# EPICS substitutions: apps/CaenHVApp/Db/CaenHV_crate11.substitutions
file "db/AS503_Chan.template" {
pattern
    {P,      H,  S,   V}
    {hchv,  11,  00,  000}
    {hchv,  11,  00,  001}
    {hchv,  11,  00,  002}
    {hchv,  11,  00,  003}
    {hchv,  11,  00,  004}
    {hchv,  11,  00,  005}
    {hchv,  11,  00,  006}
    {hchv,  11,  00,  007}
    {hchv,  11,  00,  008}
    {hchv,  11,  00,  009}
    {hchv,  11,  00,  010}
    {hchv,  11,  00,  011}
    {hchv,  11,  00,  012}
    {hchv,  11,  00,  013}
    {hchv,  11,  00,  014}
    {hchv,  11,  00,  015}
}
file "db/AS503_Chan.template" {
pattern
    {P,      H,  S,   V}
    {hchv,  11,  01, 000}
    {hchv,  11,  01, 001}
    {hchv,  11,  01, 002}
    {hchv,  11,  01, 003}
    {hchv,  11,  01, 004}
    {hchv,  11,  01, 005}
    {hchv,  11,  01, 006}
    {hchv,  11,  01, 007}
    {hchv,  11,  01, 008}
    {hchv,  11,  01, 009}
    {hchv,  11,  01, 010}
    {hchv,  11,  01, 011}
    {hchv,  11,  01, 012}
    {hchv,  11,  01, 013}
    {hchv,  11,  01, 014}
    {hchv,  11,  01, 015}
}
file "db/AS503_Chan.template" {
pattern
    {P,      H,  S,   V}
    {hchv,  11,  02, 000}
    {hchv,  11,  02, 001}
    {hchv,  11,  02, 002}
    {hchv,  11,  02, 003}
    {hchv,  11,  02, 004}
    {hchv,  11,  02, 005}
    {hchv,  11,  02, 006}
    {hchv,  11,  02, 007}
    {hchv,  11,  02, 008}
    {hchv,  11,  02, 009}
    {hchv,  11,  02, 010}
    {hchv,  11,  02, 011}
    {hchv,  11,  02, 012}
    {hchv,  11,  02, 013}
    {hchv,  11,  02, 014}
    {hchv,  11,  02, 015}
}
file "db/AS503_Chan.template" {
pattern
    {P,      H,  S,   V}
    {hchv,  11,  03, 000}
    {hchv,  11,  03, 001}
    {hchv,  11,  03, 002}
    {hchv,  11,  03, 003}
    {hchv,  11,  03, 004}
    {hchv,  11,  03, 005}
    {hchv,  11,  03, 006}
    {hchv,  11,  03, 007}
    {hchv,  11,  03, 008}
    {hchv,  11,  03, 009}
    {hchv,  11,  03, 010}
    {hchv,  11,  03, 011}
    {hchv,  11,  03, 012}
    {hchv,  11,  03, 013}
    {hchv,  11,  03, 014}
    {hchv,  11,  03, 015}
}
